PROGRAM p_MotorControl_ST
VAR
	MC_GearOutDrive1 :MC_Gearout;
	Mc_ResetServoA : MC_Reset;
	Mc_ResetServoB : MC_Reset;
	FbMc_PowerServoB :MC_Power;
	FbMc_PowerServoA :MC_Power;
	

 ServoResetOK :BYTE;
 
 jogbuttontimer :ton;
 
 //Monitor the rising edge of the ecnoder position reset function.
 
ServosReady :byte; // 	
 
// ServoEnableFallingEdge: f_trig;	
 // ServoEnableRisingEdge: r_trig;	
 // SoeResetRisingEdge :r_trig;
	st_Buffermode : MC_Buffermode;
	n_Override :INT := 100;
	SoeReset :BYTE;
	
   EncodeCalibrationRequest_RisingEdge :r_trig;
	
	b_debugSetEncoders: BOOL;
	debugging_belt: BOOL;
	BufferMode: MC_Buffermode;
	BeltForceBit: BOOL;
	state: INT; // State machine current step
	b_ServosReady: BOOL;
	b_Faulted: BOOL;
	testbool: BOOL;
	ServoDisableTimeout :Ton;
	b_DEBUG_STOP: BOOL;
	b_EncoderCalibrationRequest: BOOL;
	RequestedState: INT;
	Requested: INT;
	n_JogReq: INT;
	ServoEnableRtrig : r_trig;
	PowerEnableRtrig: r_trig;
	MoveDoneRtrig: r_trig;
	ExecuteButtonRtrig: R_trig;
	JogRtrig: R_trig;
	JogUpRtrig: R_trig;;
	JogDnRtrig: R_trig;
END_VAR

st_buffermode := MC_Aborting; // stop between moves instead of blending? see the mc_buffermode docs
jogbuttontimer.PT := T#250MS;
b_Faulted := p_faultmonitoring.b_Faulted;
Mc_ResetServoA(Axis := io.DriveAxis1, Execute := Control.b_RequestServoReset);
Mc_ResetServoB(Axis := io.DriveAxis2, Execute := Control.b_RequestServoReset);//STb
io.DriveEnable1 := Control.b_EnableServosFinal;
io.DriveEnable2 := control.b_EnableServosFinal;
MC_GearOutDrive1(Slave := io.DriveAxis2, Execute := NOT Control.b_ExecuteGearIn);
servoenablertrig(CLK := io.PowerEnabled) ;
IF servoenablertrig.q THEN
	control.b_EnableServosReq := TRUE;
END_IF

PowerEnableRtrig(CLK := Global_variables.HmiButtonData0.2) ; // power on off request handler.

IF PowerEnableRtrig.q  AND NOT b_faulted THEN // if we get a power on request, and we're not faulted, try turning on power. turn it off if it's already on.
	IF io.PowerEnabled THEN 
		io.PowerEnabled := FALSE;
		ELSE
		io.PowerEnabled := TRUE;
		END_IF
	END_IF

IF b_faulted THEN io.PowerEnabled := FALSE; END_IF; // drop power on fault.


IF NOT io.PowerEnabled THEN
	control.b_EnableServosReq := false;
END_IF

IF Control.b_RequestServoReset OR b_Faulted OR NOT IO.PowerEnabled THEN // if faulted, reset, or powered off Go to state 0
state :=0; //Reset state
END_IF 






CASE state OF 
	
0: //Faulted OR Not enabled, but stopped (intialize here)
//servo power off, disable all moves and halts.			
control.b_EnableServosFinal := FALSE; // servo power off
control.b_HaltRequest := FALSE; //
control.b_UseExternalSetpointGenerator := FALSE;
control.bAbsMoveAExecute := FALSE;
control.bAbsMoveBExecute := FALSE;
 control.b_ExecuteGearIn := FALSE;

IF control.b_EnableServosReq AND (NOT b_faulted  AND NOT safety.GLOBAL_SAFETY_NOT_OK) THEN
	state := 1; // Leave the faulted state when not faulted.
	//Control.b_RequestServoReset := TRUE;
END_IF
 
1: //ready to enable, but haven't been asked to.
	 // sit here until user enable is high // user can issue reset during this stage to help wake motors.
IF NOT p_FaultMonitoring.b_Faulted AND io.PowerEnabled THEN // 
	control.b_EnableServosFinal := TRUE; // Enable the servos if the servo request is on.
//	Control.b_RequestServoReset := FALSE;	
	ELSE
		control.b_EnableServosFinal := FALSE; // Enable the servos if the servo request is on.
		State := 0;
END_IF


IF b_ServosReady THEN state := 2; END_IF; // if the servos are all enabled, we can move to next state

2: // Turning on servos with NO Commands issued, so halt them. 
control.b_HaltRequest := TRUE;	
IF control.b_Servos_Halted AND RequestedState <> 0 THEN State := RequestedState; END_IF; 

IF control.b_EnableServosReq = FALSE THEN control.b_EnableServosFinal := FALSE; State:=0; END_IF 


state := 5;	// attempt Gear in 	


3: //Switch into SP mode
	;//Enabeld, turn off halts, turn on SP generator access to servos
	control.b_HaltRequest := FALSE;
	control.b_UseExternalSetpointGenerator := TRUE;

	IF control.b_SetpointGeneratorFault	THEN State:= 4; END_IF; //halt if setpoint generator gets an error.
	IF NOT b_ServosReady THEN state := 4; END_IF; // drop power to servos if any servo loses op mode
 

4: //Enable has been dropped, HALT! (No time delay)
	control.b_UseExternalSetpointGenerator := FALSE;
 
	control.b_HaltRequest := TRUE;
   IF control.b_Servos_Halted THEN State := 0; END_IF; //drop back to initial state when halted.
   IF NOT (control.b_EnableServosReq) THEN state := 0; END_IF;
   IF ServoDisableTimeout.Q THEN State := 0; END_IF;
   
   
   
 5://gear in 

 control.b_HaltRequest := FALSE;
 control.b_ExecuteGearIn := TRUE;
 IF P_Motorcontrol.MC_GearInA.InGear THEN 
;
 END_IF

	
40: // CSV follower.
	Control.fTargetPosA := STRING_TO_LREAL(p_textmoderead.database[Control.nPlayBackIndex]);

IF NOT (p_motorcontrol.MC_MoveAbsolute_A.Active) THEN
	control.bAbsMoveAExecute := TRUE;
	State := 41;
	END_IF;
 41:
 MoveDoneRTrig(CLK := p_motorcontrol.MC_MoveAbsolute_A.InEndVelocity OR io.DriveAxis1.Status.InPositionArea);
control.bAbsMoveAExecute := FALSE;
IF MoveDoneRTrig.Q THEN // index to next move if not at end of file.

	IF Control.nPlayBackIndex <= Control.n_RowsReadfromCsv THEN
	Control.nPlayBackIndex := Control.nPlayBackIndex +1;
	State := 40;
	ELSE State := 0; 	// quit.
	END_IF

END_IF


//IF p_motorcontrol.MC_MoveAbsolute_A.error THEN state := 110; END_IF



110: 
;
111: //reached end
	;
END_CASE

Servodisabletimeout.PT := T#1000MS;
Servodisabletimeout(IN:=(state = 4)); //.q is true 2 seconds after servo enable is no longer commanded
 
//Servo enable command sent rising edge	
//ServoEnableRisingedge(CLK:=control.b_EnableServosFinal);
// lost enable, start halt & shutdown procedure
//ServoEnableFallingedge(CLK:=(Control.b_MainCoreServoEnableReq AND control.b_EnableServosReq));

//Send halt command to NC (this is here for timing reasons)
Control.b_HaltRequestExecute := control.b_HaltRequest; // halt if requested, unless the servo system is disabled.  


// pack servo readdy bits into the servoready byte. if a Bit is true, the assosiated servo is ready to roll.
Servosready.0 := io.DriveEnabled1;
Servosready.1 := io.DriveEnabled2;

IF ServosReady = 3 THEN //if all servos ready set bool true
	b_ServosReady := TRUE;
	ELSE
	b_Servosready :=FALSE;
END_IF

Control.n_ServosHalted.0 := P_MotorControl.MC_Halt_ServoB.Done;
Control.n_ServosHalted.1 := P_MotorControl.MC_Halt_ServoA.Done;

//detect when everything is halted.
IF control.n_ServosHalted = 3 THEN // change back to 255 to watch pendulum and laser
	control.b_Servos_Halted :=TRUE;
	ELSE
	control.b_Servos_Halted :=FALSE;
END_IF


//a
	FbMc_PowerServoA(Enable		:= io.DriveEnabled1,
			Enable_Positive	:= Control.b_EnableServosFinal ,
			Enable_Negative	:= Control.b_EnableServosFinal ,
			Override		:= n_Override ,
			BufferMode		:= st_Buffermode ,
			Axis			:= io.DriveAxis1 );

//Servo B		
	FbMc_PowerServoB(Enable		:= io.DriveEnabled2,
			Enable_Positive	:= Control.b_EnableServosFinal ,
			Enable_Negative	:= Control.b_EnableServosFinal ,
			Override		:= n_Override ,
			BufferMode		:= st_Buffermode ,
			Axis			:= io.DriveAxis2 );	

			
			// when we see execute reset a bit,
			// watch rising edge for done bit blocking it with error bit?
			//set /reset bits to fill offsets byte
			//send summary

END_PROGRAM

(* stored: Version 1.1.0.1, ProductVersion 3.1.4024.4
   POU p_MotorControl_ST: Id {1948efc2-07af-4f24-8417-60a242e950fd}, SpecialFunc None *)
